ABB RobotStudio station: 2bots_1_20191130-204123.rsstn

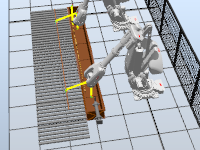
Station 2bots_1 (saved by RobotStudio 7.0.8683.559)
Controller Controller1, task T_ROB2: task frame (RAPID world) sits at (0, 1000, 0) mm in the station
Controller Controller1, task T_ROB1: task frame (RAPID world) sits at (0, 1000, 0) mm in the station
Controller Controller1
  mechanical unit ROB_1: IRB8700_550_420__01, 6 joints, base frame (0, 0, 0) mm
  mechanical unit ROB_2: IRB8700_550_420__01_2, 6 joints, base frame (0, 4000, 0) mm
Layout (positions relative to the parent item):
  - IRB8700_550_420__01 [mechanism, from Robots\IRB8700_550_420__01.rslib] at (0, 1000, 0) mm; joint values [0.0105, 0.2608, 1.1985, -3.1231, 0.4131, -1.5803] (rad or m)
  - IRB8700_550_420__01_2 [mechanism, from Robots\IRB8700_550_420__01.rslib] at (0, 5000, 0) mm; joint values [0, 0.0249, 0.9353, 0, 0.6355, 1.5708] (rad or m)
  - box [part] at (2250, 0, 0) mm, rotated rx 0 ry 0 rz 90 deg
  - Staket [part, from Downloads\f92716b2-df30-422d-9f65-0dc4c08bf145staket.rslib] at (-1500, 2000, 0) mm
  - Staket_2 [part, from Downloads\f92716b2-df30-422d-9f65-0dc4c08bf145staket.rslib] at (-1500, 0, 0) mm
  - Staket_3 [part, from Downloads\f92716b2-df30-422d-9f65-0dc4c08bf145staket.rslib] at (-1500, 4000, 0) mm
  - Staket_4 [part, from Downloads\f92716b2-df30-422d-9f65-0dc4c08bf145staket.rslib] at (-1500, 6000, 0) mm
  - Staket_5 [part, from Downloads\f92716b2-df30-422d-9f65-0dc4c08bf145staket.rslib] at (-1500, 8000, 0) mm
  - Staket_6 [part, from Downloads\f92716b2-df30-422d-9f65-0dc4c08bf145staket.rslib] at (-1500, -2000, 0) mm
  - Component1 [part] at (4000, 7000, 420) mm, rotated rx 90 ry 0 rz -90 deg
  - Gripper [mechanism, from Rar$DRa2952.43288\Gripper.rslib] at (2000, 5000, 703.2) mm, rotated rx 180 ry 0 rz 0 deg; joint values [0] (rad or m)
  - Gripper_2 [mechanism, from Rar$DRa2952.833\Gripper.rslib] at (2126.52, 1020, 394.19) mm, rotated rx -180 ry -45 rz 0 deg; joint values [0] (rad or m)
  - TUBE_ATT [smart component, from Components\Attacher.rslib]
      properties: Parent=Gripper_2; Flange=0; Child=TUBE; Mount=false; Offset=[2.5 0 3.5]; Orientation=[0 0 1.5707963267949]
  - Tube_in_box [part] at (-1000, 0, -400) mm
  - TUBE_DET [smart component, from Components\Detacher.rslib]
      properties: Child=TUBE; KeepPosition=true
  - COL_ATT_TUBE [smart component, from Components\CollisionSensor.rslib]
      properties: Object1=Gripper_2; Object2=TUBE; NearMiss=0.01; Part1=(none); Part2=(none); CollisionType=0
  - COL_TUBE_DET [smart component, from Components\CollisionSensor.rslib]
      properties: Object1=Gripper_2; Object2=Tube_in_box; NearMiss=0.1; Part1=(none); Part2=(none); CollisionType=0
  - TUBE [part] at (-25, 0, 0) mm
  - Tube_In_Place [part] at (0, 20, 0) mm
  - COL_TUBE_INPLACE [smart component, from Components\CollisionSensor.rslib]
      properties: Object1=Tube_In_Place; Object2=TUBE; NearMiss=0; Part1=(none); Part2=(none); CollisionType=0
  - PISTON1_EXPAND [smart component, from Components\LinearMover2.rslib]
      properties: Object=PISTON3; Direction=[0 0.001 0]; Distance=0.1; Duration=0.5; Reference=Global; ReferenceObject=(none)
  - PISTON1_RETRACT [smart component, from Components\LinearMover2.rslib]
      properties: Object=PISTON3; Direction=[0 -0.001 0]; Distance=0.1; Duration=0.5; Reference=Global; ReferenceObject=(none)
  - TAP1 [part] at (0, 95, 0) mm
  - Attacher [smart component, from Components\Attacher.rslib]
      properties: Parent=TUBE; Flange=0; Child=TAP1; Mount=false; Offset=[0 0 0]; Orientation=[0 0 0]
  - Detacher [smart component, from Components\Detacher.rslib]
      properties: Child=TAP1; KeepPosition=true
  - PISTON2 [part] at (0, 5850, 1740) mm, rotated rx 180 ry 0 rz 0 deg
  - PISTON2_BODY [part] at (0, 5850, 1740) mm, rotated rx 180 ry 0 rz 0 deg
  - Detacher_2 [smart component, from Components\Detacher.rslib]
      properties: Child=TAP1_3; KeepPosition=true
  - Attacher_2 [smart component, from Components\Attacher.rslib]
      properties: Parent=TUBE; Flange=0; Child=TAP1_3; Mount=false; Offset=[0 0 0]; Orientation=[0 0 0]
  - PISTON_2_RETRACT [smart component, from Components\LinearMover2.rslib]
      properties: Object=PISTON4; Direction=[0 0.001 0]; Distance=0.09; Duration=0.5; Reference=Global; ReferenceObject=(none)
  - PISTON_2_EXPAND [smart component, from Components\LinearMover2.rslib]
      properties: Object=PISTON4; Direction=[0 -0.001 0]; Distance=0.09; Duration=0.5; Reference=Global; ReferenceObject=(none)
  - PISTON3_BODY [part] at (2000, -300, 865) mm, rotated rx 180 ry 0 rz 0 deg
  - PISTON3 [part] at (2000, -200, 865) mm, rotated rx 180 ry 0 rz 0 deg
  - PISTON4_BODY [part] at (2000, 6100, 865) mm
  - PISTON4 [part] at (2000, 6040, 865) mm
  - PISTON1_HOLDER [part] at (2000, -110, 865) mm, rotated rx 180 ry 0 rz 180 deg
  - TAP1_3 [part] at (2000, 5900, 865) mm, rotated rx 180 ry 0 rz 180 deg
  - PISTON2_HOLDER [part] at (2000, 5940, 865) mm, rotated rx 180 ry 0 rz 180 deg
  - analogprogrammers [part] at (2200, 600, 0) mm, rotated rx 90 ry 0 rz 90 deg
Attachment: Gripper is attached to IRB8700_550_420__01_2 / Link6
Attachment: Gripper_2 is attached to IRB8700_550_420__01 / Link6
Attachment: TAP1 is attached to PISTON3
Attachment: TAP1_3 is attached to PISTON4
Station signals: DI Reset
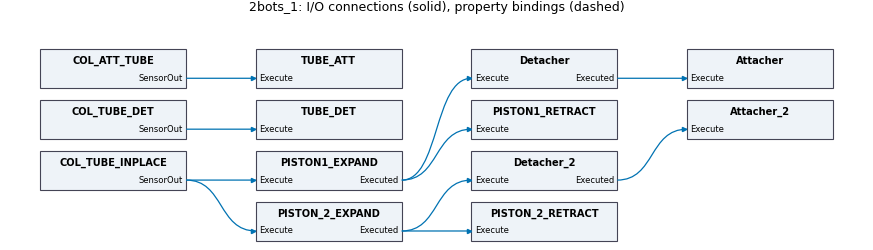
Station logic (signal -> signal, property => property):
  COL_ATT_TUBE.SensorOut -> TUBE_ATT.Execute
  COL_TUBE_DET.SensorOut -> TUBE_DET.Execute
  COL_TUBE_INPLACE.SensorOut -> PISTON1_EXPAND.Execute
  PISTON1_EXPAND.Executed -> Detacher.Execute
  Detacher.Executed -> Attacher.Execute
  PISTON1_EXPAND.Executed -> PISTON1_RETRACT.Execute
  Detacher_2.Executed -> Attacher_2.Execute
  COL_TUBE_INPLACE.SensorOut -> PISTON_2_EXPAND.Execute
  PISTON_2_EXPAND.Executed -> Detacher_2.Execute
  PISTON_2_EXPAND.Executed -> PISTON_2_RETRACT.Execute
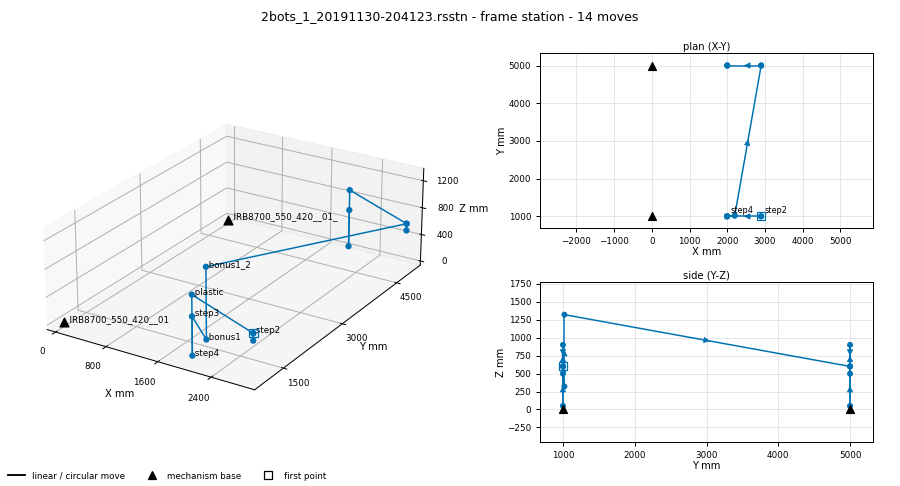
[picture p0: tool path of 2bots_1_20191130-204123.rsstn in frame station, 14 of 14 moves have a stored position in this frame; points joined in program order, loops and branches not executed]
Targets, tools, work objects and paths stored in the station, written as RAPID:
! task T_ROB1
MODULE Module1
  CONST robtarget step2:=[[2900,0,600],[0,0,1,0],[0,0,0,0],[9E+09,9E+09,9E+09,9E+09,9E+09,9E+09]];
  CONST robtarget step4:=[[2000,0,50],[0,0,1,0],[0,0,0,0],[9E+09,9E+09,9E+09,9E+09,9E+09,9E+09]];
  CONST robtarget step3:=[[2000,0,600],[0,0,1,0],[0,0,0,0],[9E+09,9E+09,9E+09,9E+09,9E+09,9E+09]];
  CONST robtarget step1:=[[2899.846169767,0.00000506,498.684966046],[0.000000008,0.000000022,1,0],[-1,0,1,0],[9E+09,9E+09,9E+09,9E+09,9E+09,9E+09]];
  CONST robtarget plastic:=[[2000,0,900],[0,0,1,0],[0,0,0,0],[9E+09,9E+09,9E+09,9E+09,9E+09,9E+09]];
  CONST robtarget bonus1:=[[2199.497474705,20,321.213203385],[0.382683432,0,0.923879533,0],[0,-2,-2,0],[9E+09,9E+09,9E+09,9E+09,9E+09,9E+09]];
  CONST robtarget bonus1_2:=[[2199.497476705,20,1321.213203385],[-0.000000001,0,1,0],[0,0,1,0],[9E+09,9E+09,9E+09,9E+09,9E+09,9E+09]];
  PROC Path_10()
    MoveL step2,v1000,z100,tGripper\WObj:=wobj0;
    MoveL step1,v1000,z100,tGripper\WObj:=wobj0;
    MoveL step2,v1000,z100,tGripper\WObj:=wobj0;
    MoveL plastic,v1000,z100,tGripper\WObj:=wobj0;
    WaitTime 2;
    MoveC step3,step4,v1000,z100,tGripper\WObj:=wobj0;
    MoveL step3,v1000,z100,tGripper\WObj:=wobj0;
    WaitTime 2;
    MoveL bonus1,v1000,z100,tGripper\WObj:=wobj0;
    MoveL bonus1_2,v1000,z100,tGripper\WObj:=wobj0;
  ENDPROC
ENDMODULE

! task T_ROB1
MODULE CalibData
  PERS tooldata tGripper:=[TRUE,[[0,0,103.2],[0.707106781,0,0,-0.707106781]],[1,[1.056741569,1.153178972,50.827393488],[1,0,0,0],0,0,0]];
ENDMODULE

! task T_ROB2
MODULE CalibData
  PERS tooldata KN240_IRB1600:=[TRUE,[[-115,0,220],[0,-0.707106781,0,0.707106781]],[4.315,[-69.777,0.103,116.319],[1,0,0,0],0.0285,0.02306,0.01111]];
  PERS tooldata tGripper:=[TRUE,[[0,0,103.2],[0.707106781,0,0,-0.707106781]],[1,[1.056741569,1.153178972,50.827393488],[1,0,0,0],0,0,0]];
ENDMODULE

! task T_ROB2
MODULE Module1
  CONST robtarget plastic:=[[2000,4000,900],[0,0,1,0],[0,0,0,0],[9E+09,9E+09,9E+09,9E+09,9E+09,9E+09]];
  CONST robtarget step1:=[[2900.846,4000,498.685],[0,0,1,0],[0,0,0,0],[9E+09,9E+09,9E+09,9E+09,9E+09,9E+09]];
  CONST robtarget step2:=[[2900,4000,600],[0,0,1,0],[0,0,0,0],[9E+09,9E+09,9E+09,9E+09,9E+09,9E+09]];
  CONST robtarget step3:=[[2000,4000,600],[0,0,1,0],[0,0,0,0],[9E+09,9E+09,9E+09,9E+09,9E+09,9E+09]];
  CONST robtarget step4:=[[2000,4000,50],[0,0,1,0],[0,0,0,0],[9E+09,9E+09,9E+09,9E+09,9E+09,9E+09]];
  PROC Path_10()
    MoveL step2,v1000,z100,tGripper\WObj:=wobj0;
    MoveL step1,v1000,z100,tGripper\WObj:=wobj0;
    MoveL step2,v1000,z100,tGripper\WObj:=wobj0;
    MoveL plastic,v1000,z100,tGripper\WObj:=wobj0;
    WaitTime 2;
    MoveC step3,step4,v1000,z100,tGripper\WObj:=wobj0;
    MoveL step3,v1000,z100,tGripper\WObj:=wobj0;
  ENDPROC
ENDMODULE

